// TwinCAT 3 PLC project _Example_Log
// ProgramVersion: 3.1.4024.0
// libraries:
//   Tc2_Standard, * (Beckhoff Automation GmbH)
//   Tc2_System, * (Beckhoff Automation GmbH)
//   Tc2_Utilities, * (Beckhoff Automation GmbH)
//   Tc3_Module, * (Beckhoff Automation GmbH)
// project tree:
//   GVLs/ GVL.TcGVL, MSG.TcGVL
//   / PlcTask.TcTTO
//   POUs/ FB_UpdateTimeStamp.TcPOU, MAIN.TcPOU, LOGGING.TcPOU
// real-time tasks:
//   TASK PlcTask: cycle T#10ms, priority 20, ADS port 350

CONFIGURATION _Example_Log
    RESOURCE PLC ON TwinCAT3
        TASK PlcTask(INTERVAL := T#10ms, PRIORITY := 20);
        PROGRAM MAIN WITH PlcTask : MAIN;
    END_RESOURCE
END_CONFIGURATION

// ---- GVLs/GVL.TcGVL
{attribute 'qualified_only'}
VAR_GLOBAL
	// Create this Folder to store log
	Log_Directory : STRING := 'C:\Users\celli\OneDrive\Desktop\TEST_LOG\PROCESS\';
END_VAR

VAR_GLOBAL PERSISTENT
	yesterday 	: STRING;
	today		: STRING;
END_VAR

// ---- GVLs/MSG.TcGVL
{attribute 'qualified_only'}
VAR_GLOBAL
	// EVENT
	EVENT_BTN				: STRING := '[BTN] ';
	EVENT_HMI				: STRING := '[HMI] ';
	EVENT_PROCESS			: STRING := '[PROCESS] ';
	
	// COMPONENT
	COMP_CYLINDER_1			: STRING := '|CYL 1|';
	COMP_CYLINDER_2			: STRING := '|CYL 2|';
	COMP_CONV_MOTOR_1		: STRING := '|Conveyor Motor|';
	
	// ACTION
	ACTION_EXTEND 			: STRING := 'CYL Extend';
	ACTION_RETRACT 			: STRING := 'CYL Retract';
	ACTION_MOTOR_RUN 		: STRING := 'Motor Run Forward';
	
	//STATUS
	STATUS_RUN				: STRING := '(Run)';
	STATUS_ACK				: STRING := '(Ack)';
	STATUS_DONE				: STRING := '(Done)';
END_VAR

// ---- POUs/MAIN.TcPOU
PROGRAM MAIN
VAR
	LogProcess		: LOGGING;
	fb_TimeStamp 	: FB_UpdateTimeStamp ();
	
	bLog_Flag		: BOOL;
	bLog_Flag1		: BOOL;
END_VAR

fb_TimeStamp();

IF bLog_Flag THEN
	LogProcess( sLogEvent	 := MSG.EVENT_PROCESS, 
	 			sLogComp	 := MSG.COMP_CONV_MOTOR_1, 
	 			sLogAction	 := MSG.ACTION_MOTOR_RUN, 
	 			sLogStatus	 := MSG.STATUS_DONE,
	 		 	blogFlag	 := TRUE);
	IF LogProcess.blog_complete OR LogProcess.blog_error THEN
		bLog_Flag 			:= FALSE;
	END_IF
END_IF

IF bLog_Flag1 THEN
	LogProcess( sLogEvent	 := MSG.EVENT_PROCESS, 
	 			sLogComp	 := MSG.COMP_CYLINDER_1, 
	 			sLogAction	 := MSG.ACTION_MOTOR_RUN, 
	 			sLogStatus	 := MSG.STATUS_DONE,
	 		 	blogFlag	 := TRUE);
	IF LogProcess.blog_complete OR LogProcess.blog_error THEN
		bLog_Flag1 			:= FALSE;
	END_IF
END_IF

END_PROGRAM

// ---- POUs/LOGGING.TcPOU
FUNCTION_BLOCK LOGGING

VAR_INPUT
	sLogEvent		: STRING;
	sLogComp		: STRING;
	sLogAction		: STRING;
	sLogStatus		: STRING;
	blogFlag		: BOOL;
END_VAR
VAR_OUTPUT
	blog_complete 	: BOOL := FALSE;
	blog_error	 	: BOOL := FALSE;
END_VAR
VAR
	fb_TimeStamp : FB_UpdateTimeStamp ();
	fbCreateDir	 : FB_CreateDir;
	fbFileOpen	 : FB_FileOpen;
	fbFileWrite	 : FB_FilePuts;
	fbFileClose	 : FB_FileClose;
	ilog_state	 : ( INIT, 
					 CREATE_DIR, 
					 FILE_OPEN,
					 WRITE_TITLE,
					 WRITE_LOG, 
					 FILE_CLOSE,
					 CLEAR, 
					 ERROR);
	
	sTextLog	 	: STRING[300];		
	sFolderName	 	: STRING;
	sLastFolderName	: STRING;
	sFileName		: STRING;
	sLastFileName 	: STRING;	
		
	sWritepLog	 : STRING[300];
	sWriteTitle	 : STRING;
	
	sInLogEvent	: STRING;
	sInLogComp	: STRING;
	sInLogAction	: STRING;
	sInLogStatus	: STRING;
	
END_VAR

IF sLogComp<>sInLogComp OR sLogAction<>sInLogAction OR sLogStatus<>sInLogStatus THEN
	sInLogEvent		:= sLogEvent;
	sInLogComp		:= sLogComp;
	sInLogAction	:= sLogAction;
	sInLogStatus	:= sLogStatus;
ELSE
	RETURN;
END_IF

sTextLog := string_concat(sInLogEvent, sInLogComp,sInLogAction,sInLogStatus);

WHILE blogFlag DO
	CASE ilog_state OF
		// INIT -------------------------------------------------------------------
		INIT:
			blog_complete	:= FALSE;
			blog_error		:= FALSE;
			ilog_state 		:= CREATE_DIR;
			fbCreateDir(bExecute:= FALSE);
	
		// CREATE_DIR -------------------------------------------------------------			
		CREATE_DIR:	
			sFolderName := CONCAT(GVL.Log_Directory, MAIN.fb_TimeStamp.SystemDate);

			IF sFolderName = sLastFolderName THEN
				ilog_state := FILE_OPEN;
				fbCreateDir(bExecute := FALSE);
				fbFileOpen(bExecute := FALSE);
			ELSE
				fbCreateDir( sPathName:= sFolderName, bExecute:= TRUE );
				IF NOT fbCreateDir.bBusy THEN
					ilog_state := FILE_OPEN;
					fbCreateDir(bExecute := FALSE);
					fbFileOpen(bExecute := FALSE);
					sLastFolderName := sFolderName;
				END_IF
			END_IF
			
		// FILE_OPEN -------------------------------------------------------------
		FILE_OPEN:
			sFileName := CONCAT(sFolderName,'\');
			sFileName := CONCAT(sFileName, MAIN.fb_TimeStamp.SystemHour);
			sFileName := CONCAT(sFileName,'.csv');
				
			fbFileOpen( sPathName	:= sFileName, 
						nMode		:= FOPEN_MODEAPPEND, 
						bExecute	:= TRUE, 
						hFile=>);
			IF fbFileOpen.bError THEN
				ilog_state := ERROR;
				fbFileOpen(bExecute := FALSE);
				fbFileWrite(bExecute := FALSE);
			ELSIF NOT fbFileOpen.bBusy THEN
				ilog_state := WRITE_TITLE;
				fbFileOpen(bExecute := FALSE);
				fbFileWrite(bExecute := FALSE);
			END_IF
			
		// WRITE_TITLE -------------------------------------------------------------
		WRITE_TITLE:
			IF sLastFileName <> sFileName THEN	
				sWriteTitle := CONCAT('$n','Time Stamp');
				sWriteTitle := CONCAT(sWriteTitle,',');
				sWriteTitle := CONCAT(sWriteTitle,'Event');
				sWriteTitle := CONCAT(sWriteTitle,',');
				sWriteTitle := CONCAT(sWriteTitle,'Component');
				sWriteTitle := CONCAT(sWriteTitle,',');
				sWriteTitle := CONCAT(sWriteTitle,'Action');
				sWriteTitle := CONCAT(sWriteTitle,',');
				sWriteTitle := CONCAT(sWriteTitle,'Status');
				
				fbFileWrite ( hFile:=fbFileOpen.hFile,
								sLine:=sWriteTitle,
								bExecute:=TRUE);
				IF fbFileWrite.bError THEN
					ilog_state := ERROR;
					fbFileWrite(bExecute := FALSE);
					fbFileClose(bExecute := FALSE);
				ELSIF NOT fbFileWrite.bBusy THEN
					ilog_state := WRITE_LOG;
					fbFileWrite(bExecute := FALSE);
					fbFileClose(bExecute := FALSE);
					sLastFileName := sFileName;
				END_IF
			ELSE
				ilog_state := WRITE_LOG;
			END_IF

		// WRITE_LOG -------------------------------------------------------------
		WRITE_LOG:	
			sWritepLog := sTextLog;
			
			fbFileWrite ( 	hFile		:=fbFileOpen.hFile,
							sLine		:=sWritepLog,
							bExecute	:=TRUE);
			IF fbFileWrite.bError THEN
				ilog_state := ERROR;
				fbFileWrite(bExecute := FALSE);
				fbFileClose(bExecute := FALSE);
			ELSIF NOT fbFileWrite.bBusy THEN
				ilog_state := FILE_CLOSE;
				fbFileWrite(bExecute := FALSE);
				fbFileClose(bExecute := FALSE);
			END_IF
			
		// FILE_CLOSE -------------------------------------------------------------
		FILE_CLOSE:			
			fbFileClose( hFile		:=fbFileOpen.hFile,
						 bExecute	:=TRUE);
			IF fbFileClose.bError THEN
				ilog_state := ERROR;
				fbFileClose(bExecute := FALSE);
			ELSIF NOT fbFileClose.bBusy THEN
				ilog_state := CLEAR;
				fbFileClose(bExecute := FALSE);
			END_IF
			
		// CLEAR -------------------------------------------------------------	
		CLEAR:
			blog_complete	:= TRUE;
			blogFlag		:= FALSE;
			ilog_state 		:= INIT;
				
		// ERROR -------------------------------------------------------------	
		ERROR:
			blog_error		:= TRUE;
			blogFlag		:= FALSE;
			ilog_state 		:= INIT;
	END_CASE
END_WHILE

METHOD string_concat : STRING(300)
VAR_INPUT
	text1	: STRING;
	text2	: STRING;
	text3	: STRING;
	text4	: STRING;
END_VAR
VAR
	Con_String : String(300);
END_VAR
Con_String := CONCAT('$n', MAIN.fb_TimeStamp.FullSystemTime);
Con_String := CONCAT(Con_String, ' , ');
Con_String := CONCAT(Con_String, text1);
Con_String := CONCAT(Con_String, ' , ');
Con_String := CONCAT(Con_String, text2);
Con_String := CONCAT(Con_String, ' , ');
Con_String := CONCAT(Con_String, text3);
Con_String := CONCAT(Con_String, ' , ');
Con_String := CONCAT(Con_String, text4);

string_concat := Con_String;
END_METHOD

END_FUNCTION_BLOCK

// ---- POUs/FB_UpdateTimeStamp.TcPOU
FUNCTION_BLOCK FB_UpdateTimeStamp
VAR_INPUT
END_VAR
VAR_OUTPUT
	FullSystemTime	: STRING;
	SystemDate		: STRING;
	SystemTime		: STRING;
	SystemHour		: STRING;
	timeValid		: BOOL;
END_VAR
VAR
	fb_LocalTime	 : FB_LocalSystemTime;
	dayNum		: UINT;
	today 		: STRING;
END_VAR

//  --------------------------------------------------------------- Initialize
	fb_LocalTime(
			sNetID:= , 
			bEnable:= TRUE , 
			dwCycle:= 1, 
			dwOpt:= , 
			tTimeout:= ,
			bValid=> timeValid, 
			systemTime=> , 
			tzID=> );
			
//  --------------------------------------------------------------- Set system time	
	IF fb_localTime.bValid THEN
		FullSystemTime 	:= SYSTEMTIME_TO_STRING(fb_LocalTime.systemTime);
		
		SystemDate		:= WORD_TO_STRING(fb_LocalTime.systemTime.wYear);
		SystemDate		:= CONCAT(SystemDate, '.');
		SystemDate		:= CONCAT(SystemDate, WORD_TO_STRING(fb_LocalTime.systemTime.wMonth));
		SystemDate		:= CONCAT(SystemDate, '.');
		SystemDate		:= CONCAT(SystemDate, WORD_TO_STRING(fb_LocalTime.systemTime.wDay));
		Today			:= SystemDate;
		
		SystemTime		:= WORD_TO_STRING(fb_LocalTime.systemTime.wHour);
		SystemTime		:= CONCAT(SystemTime, ':');
		SystemTime		:= CONCAT(SystemTime, WORD_TO_STRING(fb_LocalTime.systemTime.wMinute));
		SystemTime		:= CONCAT(SystemTime, ':');
		SystemTime		:= CONCAT(SystemTime, WORD_TO_STRING(fb_LocalTime.systemTime.wSecond));
		
		SystemHour		:= WORD_TO_STRING(fb_LocalTime.systemTime.wHour);
	END_IF

END_FUNCTION_BLOCK
